# EPICS substitutions: hugo/source/examples/test/el7332/ecmcEL7332_volts.substitutions
file "ecmcEcSlave.template"
{
  pattern {}
          {}
}

# All fields related to velocity scaling and alarms
file "ecmcEL7332-chX.template"
{
  pattern {CH_ID, LINR,    ESLO,           EOFF,   EGU,     PREC, LOW, LOLO, HIGH, HIHI, HYST, LLSV,       LSV,        HSV,        HHSV      }
          {1      "SLOPE", 0.000732421875, 0,      "Volt",  0,    0,   0,    0,    0,    0,    "NO_ALARM", "NO_ALARM", "NO_ALARM", "NO_ALARM"}
          {2      "SLOPE", 0.000732421875, 0,      "Volt",  0,    0,   0,    0,    0,    0,    "NO_ALARM", "NO_ALARM", "NO_ALARM", "NO_ALARM"}
}
